FUNCTION_BLOCK FB_PumpGrundfosCM EXTENDS FB_Actor2Point
VAR
	//I/O Links
	bSetStatusOn_OUT 	AT %Q* : BOOL := FALSE;
END_VAR

METHOD SetState_BO : BOOL
VAR_INPUT
END_VAR
//output
bSetStatusOn_OUT := bSetStatusOn;
END_METHOD

END_FUNCTION_BLOCK

(* stored: Version 1.1.0.1, ProductVersion 3.1.4024.10
   POU FB_PumpGrundfosCM: Id {9e7f7a5e-42fe-4cc1-ac2a-50bb2a199a17}, SpecialFunc None
   Method SetState_BO: Id {0a9f2f79-143f-430a-a6d8-599f4481d4cf} *)
